PROGRAM EnOcean
VAR
	KL6581								:		FB_KL6581;
	
	KL6021FB							:		FB_EnOceanReceive;
	
	EnoceanData							:		ST_EnOceanReceivedData;
	STEnOceanInData		AT %I*			:		ST_EnOceanInData;
	STEnOceanOutData	AT %Q* 			:		ST_EnOceanOutData;
	
	//EnOcean Socket FBs
	fbXplanarScreenPower				:		FB_Send_RPS_Switch; //KL6581 Send Enocen Signals
	
	OpenTennisHMI						:		TON :=(PT := T#2S);;
	TennisHMIOpened						: 		BOOL;	
	
	TEST : ARRAY [0..3] OF BYTE;
	
	i: INT;
	
	AllWindowsClosed				:	bool;
	
	ctudCountWindows				:	ARRAY [0..5] OF CTUD;
	numberOfWindowsOpenTemp			:	ARRAY [0..5] OF WORD;
	totalNumberOfWindowsOpen		:	WORD;
	
	
END_VAR

//FB_KL6581 - Control EnOcean Terminal for transmitting 
KL6581(bInit:=TRUE, nIdx := , stKL6581_in:=stKL6581InData, stKL6581_out:= stKL6581OutData, str_KL6581=> EnOceanComms );
//FB_EnOceanReceive - Control EnOcean Receiver KL6021
KL6021FB(bEnable:= TRUE, stEnOceanReceivedData=> EnoceanData, stEnOceanInData:= STEnOceanInData, stEnOceanOutData:= STEnOceanOutData);	


// Collect all switch data
FOR i := 0 TO 3 DO
	FBEnOceanPTM200[i](
		bEnable:= TRUE, 
		bSwitches =>  ,
		nTransmitterId:= EnoceanTransmitterID[i], 
		stEnOceanReceivedData:= EnoceanData);
END_FOR

FOR i := 0 TO 5 DO	
	FBEnOceanSTM250[i](
		bEnable:= TRUE, 
		nTransmitterId:=EnoceanTransmitterIDWindows[i] , 
		stEnOceanReceivedData:= EnoceanData, 
		bState=> );
END_FOR


//Switches
PTM200StrippedTables[0].Signal := FBEnOceanPTM200[0].bSwitches[0]; // Board Room Bottom Right Off
PTM200StrippedTables[1].Signal := FBEnOceanPTM200[0].bSwitches[1]; // Board Room Bottm Left Off 
PTM200StrippedTables[2].Signal := FBEnOceanPTM200[0].bSwitches[2]; // Board Room Top Right On
PTM200StrippedTables[3].Signal := FBEnOceanPTM200[0].bSwitches[3]; // Board Room Top Left On 
PTM200StrippedTables[4].Signal := FBEnOceanPTM200[1].bSwitches[0]; // Staff Room Bottom Right Off
PTM200StrippedTables[5].Signal := FBEnOceanPTM200[1].bSwitches[1]; // Staff Room Bottom Left Off
PTM200StrippedTables[6].Signal := FBEnOceanPTM200[1].bSwitches[2]; // Staff Room Top Right On
PTM200StrippedTables[7].Signal := FBEnOceanPTM200[1].bSwitches[3]; // Staff Room Top Left On
PTM200StrippedTables[8].Signal := FBEnOceanPTM200[2].bSwitches[0]; //Floating Switch 
PTM200StrippedTables[9].Signal := FBEnOceanPTM200[2].bSwitches[1]; //Floating Switch 
PTM200StrippedTables[10].Signal := FBEnOceanPTM200[2].bSwitches[2]; //Floating Switch 
PTM200StrippedTables[11].Signal := FBEnOceanPTM200[2].bSwitches[3]; //Floating Switch 
PTM200StrippedTables[12].Signal := FBEnOceanPTM200[3].bSwitches[0]; //Tennis Table Left Bottom 
PTM200StrippedTables[13].Signal := FBEnOceanPTM200[3].bSwitches[1]; //Tennis Table Right Bottom  
PTM200StrippedTables[14].Signal := FBEnOceanPTM200[3].bSwitches[2]; //Tennis Table Left Top  
PTM200StrippedTables[15].Signal := FBEnOceanPTM200[3].bSwitches[3]; //Tennis Table Right Top  


//Window States
PTM250WindowSensor[0] := FBEnOceanSTM250[0].bState;
PTM250WindowSensor[1] := FBEnOceanSTM250[1].bState;
PTM250WindowSensor[2] := FBEnOceanSTM250[2].bState; //Window nearest big tele
PTM250WindowSensor[3] := FBEnOceanSTM250[3].bState; //Window nearest coffee machine
PTM250WindowSensor[4] := FBEnOceanSTM250[4].bState; //Window behind Alan's desk
PTM250WindowSensor[5] := FBEnOceanSTM250[5].bState; //Window next to big whiteboard

AllWindowsClosed := PTM250WindowSensor[0] AND PTM250WindowSensor[1] AND PTM250WindowSensor[2] AND PTM250WindowSensor[3] AND PTM250WindowSensor[4] AND PTM250WindowSensor[5];

//Count Open Windows for Dashboard Display
ctudCountWindows[0](
	CU:= NOT PTM250WindowSensor[0], 
	CD:= PTM250WindowSensor[0], 
	PV:= 20, 
	CV=> numberOfWindowsOpenTemp[0]);
	
ctudCountWindows[1](
	CU:= NOT PTM250WindowSensor[1], 
	CD:= PTM250WindowSensor[1], 
	PV:= 20, 
	CV=> numberOfWindowsOpenTemp[1]);
	
ctudCountWindows[2](
	CU:= NOT PTM250WindowSensor[2], 
	CD:= PTM250WindowSensor[2], 
	PV:= 20, 
	CV=> numberOfWindowsOpenTemp[2]);	
	
ctudCountWindows[3](
	CU:= NOT PTM250WindowSensor[3], 
	CD:= PTM250WindowSensor[3], 
	PV:= 20, 
	CV=> numberOfWindowsOpenTemp[3]);

ctudCountWindows[4](
	CU:= NOT PTM250WindowSensor[4], 
	CD:= PTM250WindowSensor[4], 
	PV:= 20, 
	CV=> numberOfWindowsOpenTemp[4]);

ctudCountWindows[5](
	CU:= NOT PTM250WindowSensor[5], 
	CD:= PTM250WindowSensor[5], 
	PV:= 20, 
	CV=> numberOfWindowsOpenTemp[5]);
	
totalNumberOfWindowsOpen := (numberOfWindowsOpenTemp[0] + 
								numberOfWindowsOpenTemp[1] + 
								numberOfWindowsOpenTemp[2] + 
								numberOfWindowsOpenTemp[3] + 
								numberOfWindowsOpenTemp[4] +
								numberOfWindowsOpenTemp[5]);
	
//Collect Switch Data to be collected by CX8090 via ADS READ
(*BlindCommandTable[0] := BOOL_TO_UINT(FBEnOceanPTM200[0].bSwitches[0]); 
BlindCommandTable[1] := BOOL_TO_UINT(FBEnOceanPTM200[0].bSwitches[1]); 
BlindCommandTable[2] := BOOL_TO_UINT(FBEnOceanPTM200[0].bSwitches[2]); 
BlindCommandTable[3] := BOOL_TO_UINT(FBEnOceanPTM200[0].bSwitches[3]);  
BlindCommandTable[4] := BOOL_TO_UINT(FBEnOceanPTM200[1].bSwitches[0]); 
BlindCommandTable[5] := BOOL_TO_UINT(FBEnOceanPTM200[1].bSwitches[1]);  
BlindCommandTable[6] := BOOL_TO_UINT(FBEnOceanPTM200[1].bSwitches[2]); 
BlindCommandTable[7] := BOOL_TO_UINT(FBEnOceanPTM200[1].bSwitches[3]); 
BlindCommandTable[8] := BOOL_TO_UINT(FBEnOceanPTM200[2].bSwitches[0]); 
BlindCommandTable[9] := BOOL_TO_UINT(FBEnOceanPTM200[2].bSwitches[1]); 
BlindCommandTable[10] := BOOL_TO_UINT(FBEnOceanPTM200[2].bSwitches[2]); 
BlindCommandTable[11] := BOOL_TO_UINT(FBEnOceanPTM200[2].bSwitches[3]);  	*)

//Transmit KL6581

//Screen control test ///////////////////////////////////////////////////////////////////////////////////////
//not used for screen anymore - used for display cabinet light
fbXplanarScreenPower(
	bStart:= , 
	by_Node:= 1, 
	bData:= , 
	nRockerID:= 0, 
	nEnOceanID:= 22, 
	str_KL6581:= KL6581.str_KL6581, 
	bBusy=> , 
	bError=> , 
	iErrorID=> );
	
	IF NOT fbXplanarScreenPower.bBusy AND fbXplanarScreenPower.bStart THEN
		fbXplanarScreenPower.bStart := FALSE;
	END_IF

IF xXplanarScreenPowerOn THEN //not used for screen anymore - used for display cabinet light
	fbXplanarScreenPower.bStart := TRUE;
	fbXplanarScreenPower.bData := TRUE;
	xXplanarScreenPowerOn := FALSE;
END_IF

IF xXplanarScreenPowerOff THEN //not used for screen anymore - used for display cabinet light
	fbXplanarScreenPower.bStart := TRUE;
	fbXplanarScreenPower.bData := FALSE;
	xXplanarScreenPowerOff := FALSE;
END_IF


///////////////////////////////////////////////////////////////////////////////////////////////////////////	
TableTennisSwitchHandling();

ACTION TableTennisSwitchHandling:
IF PTM200StrippedTables[12].Signal THEN  // hold in to turn off all before going home
	
	OpenTennisHMI.IN := TRUE;		
	IF OpenTennisHMI.Q THEN
		OpenTennisHMI.IN := FALSE;	
		TennisHMIOpened := TRUE;
	END_IF	
				
END_IF
END_ACTION

END_PROGRAM

(* stored: Version 1.1.0.1, ProductVersion 3.1.4024.12
   POU EnOcean: Id {3421a756-9055-48df-be7a-ba703cf96ec3}, SpecialFunc None
   Action TableTennisSwitchHandling: Id {5f929d36-fa5b-4b95-b11c-585dbc243666} *)
